INTERFACE I_Timestamp

METHOD PUBLIC IsDurationElapsed : BOOL
VAR_INPUT
	Duration : TIME;
END_VAR
END_METHOD

PROPERTY PUBLIC TimeSince : TIME
GET
END_GET
END_PROPERTY

END_INTERFACE

(* stored: Version 1.1.0.1, ProductVersion 3.1.4026.13
   Itf I_Timestamp: Id {5aee1d44-eb3a-48f1-8ae4-f77dd1bcb7ab}
   Method IsDurationElapsed: Id {796f3d21-af4f-4f57-90c1-6e38d9d25b5b}
   Property TimeSince: Id {eec676a0-5ca7-4377-bdb2-4bf763450052}
   Get Get: Id {9abbd0ae-ec6d-425f-968f-9c20dd89f1f6} *)
